TYPE "PLCtoMES_Common"
VERSION : 0.1
   STRUCT
      "P-HeartBeat" : Bool;
      "P-AtPreStop" : Bool;
      "P-AtPro" : Bool;
      "P-AtWork" : Bool;
      "P-EquipStatus" : Byte;
      "P-EquipMode" : Byte;
      "P-BuffQTY" : Array[1..10] of DInt;
      Reserve : Array[1..155] of Byte;
   END_STRUCT;

END_TYPE

